PROGRAM MAIN
VAR
    Child : FB_Child;
END_VAR

END_PROGRAM

(* stored: Version 1.1.0.1, ProductVersion 3.1.4024.3
   POU MAIN: Id {bc31b9c8-022c-43ef-a179-ed9aa5d910be}, SpecialFunc None *)
